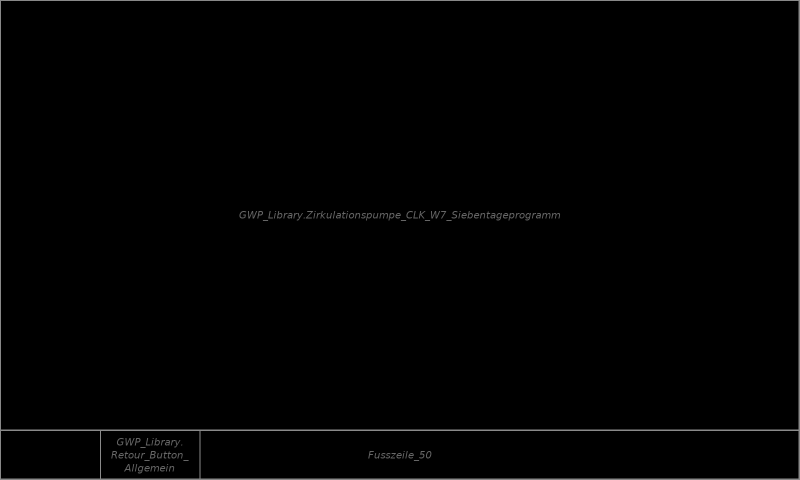
VISUALIZATION Zirkulationspumpe_CLK_W7_Siebentageprogramm  // 800x480
    Frame (0,0 800x430)
        shows GWP_Library.Zirkulationspumpe_CLK_W7_Siebentageprogramm(FB_CLK_W7 := Main.Zirk_Pumpe_0.CLK_W7_0)
    Group (0,430 800x50)
        Frame (0,0 800x50)
            shows Fusszeile_50()
        Frame (100,0 100x50)
            shows GWP_Library.Retour_Button_Allgemein()
END_VISUALIZATION

(* stored: Version 1.1.0.1, ProductVersion 3.1.4022.6
   Visu Zirkulationspumpe_CLK_W7_Siebentageprogramm: Id {24e4901d-e254-4384-9db1-e1f328a98a4d} *)
